// TIA Portal V20 export
TYPE "DigValFF"
   STRUCT
      Value : Bool;   // Value
      InternalUseBit1 { ExternalAccessible := 'False'; ExternalVisible := 'False'; ExternalWritable := 'False'} : Bool;   // Reserved / ByPass
      InternalUseBit2 { ExternalAccessible := 'False'; ExternalVisible := 'False'; ExternalWritable := 'False'} : Bool;   // Reserved
      InternalUseBit3 { ExternalAccessible := 'False'; ExternalVisible := 'False'; ExternalWritable := 'False'} : Bool;   // Reserved
      InternalUseBit4 { ExternalAccessible := 'False'; ExternalVisible := 'False'; ExternalWritable := 'False'} : Bool;   // Reserved
      InternalUseBit5 { ExternalAccessible := 'False'; ExternalVisible := 'False'; ExternalWritable := 'False'} : Bool;   // Reserved
      InternalUseBit6 { ExternalAccessible := 'False'; ExternalVisible := 'False'; ExternalWritable := 'False'} : Bool;   // Reserved
      InternalUseBit7 { ExternalAccessible := 'False'; ExternalVisible := 'False'; ExternalWritable := 'False'} : Bool;   // Reserved
      ST : Byte := BYTE#16#FF;   // Signal status / Signal Status
   END_STRUCT;
END_TYPE
